FUNCTION_BLOCK CM_Sensor2State
VAR_INPUT
	sensorInput : BOOL;
END_VAR
VAR_OUTPUT
	sensoroutput : BOOL;
END_VAR
VAR_IN_OUT
	Ctrl_CM_Sensor2State : Udt_CM_Sensor2State; 
END_VAR
VAR
END_VAR

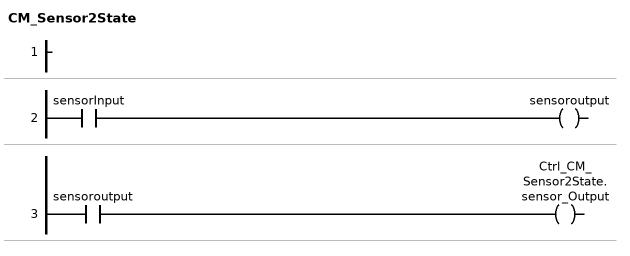
// NETWORK 1

// NETWORK 2
sensoroutput := sensorInput;

// NETWORK 3
Ctrl_CM_Sensor2State.sensor_Output := sensoroutput;

END_FUNCTION_BLOCK

(* stored: Version 1.1.0.1, ProductVersion 3.1.4024.13
   POU CM_Sensor2State: Id {c09dee76-f170-4285-b592-7fe795596600}, SpecialFunc None *)
